FUNCTION_BLOCK FB_McAxisCtrl EXTENDS FB_McAxis IMPLEMENTS I_McAxis
VAR
  _eCheck                   : E_CHECK_STATE;  // pointer check

  _eAxisCycle,                                // cyclic AXIS_REF() and MC_Power check
  _eInit                    : E_PROGRESS;     // axis startup and init, get encoder type, get axis name, get device name

  _nAxisIndex               : UINT;           // know thyself
  _rTargetWindow            : LREAL := 0.1;   // TODO: get that from NC

  // pointers to all; access required for coupling; access by index
  _Axes                     : REFERENCE TO ARRAY[1..PLC_CONSTANT.MAX_AXIS] OF AXIS_REF;

  _Ctrl                     : POINTER TO ARRAY[1..PLC_CONSTANT.MAX_AXIS] OF ST_AXIS_CTRL;    // contains command to be executed
  _State                    : POINTER TO ARRAY[1..PLC_CONSTANT.MAX_AXIS] OF ST_AXIS_STATE;   // mirrors command with added result

  _Info                     : POINTER TO ARRAY[1..PLC_CONSTANT.MAX_AXIS] OF ST_AXIS_INFO;    // axis state and position data to read from
  _Data                     : POINTER TO ARRAY[1..PLC_CONSTANT.MAX_AXIS] OF ST_MOVE_DATA;    // structure for cyclic interface

  _NcParameterWrt           : POINTER TO ARRAY[1..PLC_CONSTANT.MAX_AXIS] OF ST_NC_PARAMETER; // W struct for a single parameter
  _NcParameterRd            : POINTER TO ARRAY[1..PLC_CONSTANT.MAX_AXIS] OF ST_NC_PARAMETER; // R struct for a single parameter
  _HomeParameter            : POINTER TO ARRAY[1..PLC_CONSTANT.MAX_AXIS] OF ST_HOMING;       // homing parameter for each axis

  _GearInParameter          : POINTER TO ARRAY[1..PLC_CONSTANT.MAX_AXIS] OF ST_GEAR_IN;      // Master Indices, dyn constraints for simple GearIn

  _MotionOptions            : POINTER TO ARRAY[1..PLC_CONSTANT.MAX_AXIS] OF ST_MOTION_OPTIONS;


  // local copies of command
  _eCtrl,
  _eCtrlOld                       : E_AXIS_CTRL;

  // Last handled NC Axis parameter to write
  _eParameterNrWrite              : Tc2_MC2.MC_AxisParameter;
  _rParameterWrtValue             : LREAL;

  // Last handled NC Axis parameter to read
  _eParameterNrRead               : Tc2_MC2.MC_AxisParameter;
  _rParameterReadValue            : LREAL;

  // execution state
  _eResult                        : E_PROGRESS;   // result of execution state
  _eResultOld                     : E_PROGRESS;   // old result for detecting change
  _eState                         : E_AXIS_STATE; // execution state

  // calibration options with limit switches and simulation
  _bCalibrationCam                : BOOL;

  // mapping inputs
  _bLimitMin,
  _bLimitMax,
  _bCalibrationInput     AT %I*   : BOOL;


  // placeholder dummies in case count of Multimaster ases <> 4
  {attribute 'hide'}
  _MultiMasterDummyRef            : ARRAY[1..4] OF AXIS_REF;

  _fbGearOut                      : Tc2_MC2.MC_GearOut;
  _fbGearIn                       : Tc2_MC2.MC_GearIn;
  _fbGearInMultiMaster            : Tc2_MC2.MC_GearInMultiMaster;
END_VAR

IF NOT Check() THEN RETURN; END_IF
//-----------------------------------------------------------------------------
// check _HomeParameter for calibration input options
//-----------------------------------------------------------------------------
_bCalibrationCam                    := GetCalibrationCam();
CalibrationCam                      := ADR(_bCalibrationCam);
//-----------------------------------------------------------------------------
//-----------------------------------------------------------------------------
Override                            := _Data^[_nAxisIndex].rOverride;
//-----------------------------------------------------------------------------
//-----------------------------------------------------------------------------
// cyclic call to MC_Power and AXIS_REF()
//-----------------------------------------------------------------------------
_eAxisCycle                         := Cycle();
//-----------------------------------------------------------------------------
//-----------------------------------------------------------------------------
// get command from outside world
//-----------------------------------------------------------------------------
_eCtrl                              := _Ctrl^[_nAxisIndex].eCtrl;
//-----------------------------------------------------------------------------
//-----------------------------------------------------------------------------
//  OnChange react to command
//-----------------------------------------------------------------------------
IF (_eCtrl <> _eCtrlOld)
THEN
  // get busy
  _eState                           := Cmd(_eCtrl); // get execution state for command
  _eCtrlOld                         := _eCtrl;
  LogControl();
END_IF
//-----------------------------------------------------------------------------
//-----------------------------------------------------------------------------
//  execution state for command
//-----------------------------------------------------------------------------
CASE _eState
OF
  E_AXIS_STATE.AXIS_INIT:
    //-------------------------------------------------------------------------
    // axis always requires one init from outside world at startup
    // _eInit has to be valid for other commands to be accepted in Cmd(_eCtrl)
    _eInit := _eResult              := AxisInit(TRUE);

  E_AXIS_STATE.AXIS_NO_INIT:
    //-------------------------------------------------------------------------
    // we are here because you sent a command before having done AXIS_INIT
    _eResult                        := E_PROGRESS.ERROR;

  E_AXIS_STATE.AXIS_DISABLE:
    _eResult                        := AxisDisable(TRUE);

  E_AXIS_STATE.AXIS_ENABLE:
    _eResult                        := AxisEnable(TRUE);

  E_AXIS_STATE.AXIS_IDLE:
    _eResult                        := AxisIdle(TRUE);

  E_AXIS_STATE.AXIS_HOME:
    _eResult                        := AxisHome(TRUE);

  E_AXIS_STATE.AXIS_MOVE_POS:
    _eResult                        := AxisMoveToPosition(TRUE, _Data^[_nAxisIndex]);

  E_AXIS_STATE.AXIS_MOVE_VELO:
    _eResult                        := AxisMoveVelocity(TRUE, _Data^[_nAxisIndex]);

  E_AXIS_STATE.AXIS_RESET:
    _eResult                        := AxisReset(TRUE);

  E_AXIS_STATE.AXIS_HALT:
    _eResult                        := AxisHalt(TRUE, _Data^[_nAxisIndex]);

  E_AXIS_STATE.AXIS_STOP:
    _eResult                        := AxisStop(TRUE, _Data^[_nAxisIndex]);

  E_AXIS_STATE.AXIS_MOVE_BUFFER:
    _eResult                        := AxisBufferPos(TRUE, _Data^[_nAxisIndex]);

  E_AXIS_STATE.AXIS_MOVE_BUFFER_VELO:
    _eResult                        := AxisBufferVelo(TRUE, _Data^[_nAxisIndex]);

  E_AXIS_STATE.AXIS_PARAMETER_READ:
    _eResult                        := AxisParameterRead(TRUE, _NcParameterRd^[_nAxisIndex].ParameterNumber);

  E_AXIS_STATE.AXIS_PARAMETER_WRITE:
    _eResult                        := AxisParameterWrite(TRUE, _NcParameterWrt^[_nAxisIndex].ParameterNumber);

  E_AXIS_STATE.AXIS_PARAMETER_WRITE_PERSISTENT:
    _eResult                        := AxisParameterWritePersistent(TRUE, _NcParameterWrt^[_nAxisIndex].ParameterNumber);

  E_AXIS_STATE.AXIS_GEAR_IN:
    _eResult                        := AxisGearIn(TRUE);

  E_AXIS_STATE.AXIS_GEAR_OUT:
    _eResult                        := AxisGearOut(TRUE);

  E_AXIS_STATE.AXIS_GEAR_IN_MULTIMASTER:
    _eResult                        := AxisGearInMultiMaster(TRUE);

ELSE
  IF (_eCtrl > E_AXIS_CTRL.AXIS_NULL)
  THEN
    _eResult                          := E_PROGRESS.NOT_EXIST;
    _Info^[_nAxisIndex].bError        := TRUE;
  ELSE
    _eResult                          := E_PROGRESS.INVALID;
  END_IF
END_CASE
//-----------------------------------------------------------------------------
//-----------------------------------------------------------------------------
//  OnChange of execution state result
//    - log result and clear error number on interface
//-----------------------------------------------------------------------------
IF (_eResult <> _eResultOld)
THEN
  LogResult();
  _Info^[_nAxisIndex].nErrorId      := 0;
  _eResultOld                       := _eResult;
END_IF
//-----------------------------------------------------------------------------
//-----------------------------------------------------------------------------
// Check AxisInit
//-----------------------------------------------------------------------------
IF NOT (_eInit = E_PROGRESS.DONE)
THEN
  _Info^[_nAxisIndex].bReady        := FALSE;
ELSE
  _Info^[_nAxisIndex].bReady        := _AxisRef.Status.ControlLoopClosed AND
                                       (NOT _AxisRef.Status.Error)       AND 
                                       (NOT _AxisRef.Status.Moving);
END_IF
//-----------------------------------------------------------------------------
//  execution state result error
//-----------------------------------------------------------------------------
CASE _eResult
OF
  E_PROGRESS.ERROR:
    _Info^[_nAxisIndex].bReady      := FALSE;
    _Info^[_nAxisIndex].bError      := TRUE;
    _Info^[_nAxisIndex].nErrorId    := ErrorId;
END_CASE
//-----------------------------------------------------------------------------
// execution state result to interface
//-----------------------------------------------------------------------------
_State^[_nAxisIndex].eState       := _eState + _eResult;
//-----------------------------------------------------------------------------
// encoder type (enum)
//-----------------------------------------------------------------------------
_State^[_nAxisIndex].eAxisEncoder := EncoderType;
//-----------------------------------------------------------------------------
// _stState.[nAxisIndex].eState is overridden by MC_Power.bError
//  _eAxisCycle := Cycle() is called at the top; checks MC_Power.bError
//  MC_Power.bError requires e_AXIS_CTRL.AXIS_RESET in order to clear
//-----------------------------------------------------------------------------
CASE _eAxisCycle
OF
  E_PROGRESS.ERROR:
    _Info^[_nAxisIndex].bReady      := FALSE;
    _Info^[_nAxisIndex].bError      := TRUE;
    _State^[_nAxisIndex].eState   := _eState + _eAxisCycle;
END_CASE
//-----------------------------------------------------------------------------
// Check ControlLoop
//-----------------------------------------------------------------------------
IF _AxisRef.Status.ControlLoopClosed
THEN
  _Info^[_nAxisIndex].bEnabled      := TRUE;
ELSE
  _Info^[_nAxisIndex].bEnabled      := FALSE;
END_IF
//-----------------------------------------------------------------------------
_Info^[_nAxisIndex].bStandstill     := _AxisRef.Status.NotMoving;
//-----------------------------------------------------------------------------
_Info^[_nAxisIndex].rActPos         := _AxisRef.NcToPlc.ActPos;
_Info^[_nAxisIndex].rActVelo        := _AxisRef.NcToPlc.ActVelo;
_Info^[_nAxisIndex].rPosDiff        := _AxisRef.NcToPlc.PosDiff;
//-----------------------------------------------------------------------------
IF (_Info^[_nAxisIndex].rActPos < _Data^[_nAxisIndex].rSetPos + _rTargetWindow) AND
   (_Info^[_nAxisIndex].rActPos > _Data^[_nAxisIndex].rSetPos - _rTargetWindow) AND
    _Info^[_nAxisIndex].bStandstill
THEN
  _Info^[_nAxisIndex].bInTarget     := TRUE;
ELSE
  _Info^[_nAxisIndex].bInTarget     := FALSE;
END_IF
//-----------------------------------------------------------------------------
// copy CoupleState from axis
//-----------------------------------------------------------------------------
_Info^[_nAxisIndex].dwCoupleState   := _AxisRef.NcToPlc.CoupleState;
//-----------------------------------------------------------------------------
//-----------------------------------------------------------------------------
// copy NC AxisId from axis
//-----------------------------------------------------------------------------
_Info^[_nAxisIndex].nNcAxisId       := _AxisRef.NcToPlc.AxisId;
//-----------------------------------------------------------------------------

PROPERTY Axes : reference TO ARRAY[1..PLC_CONSTANT.MAX_AXIS] OF AXIS_REF
SET
_Axes := Axes;
END_SET
END_PROPERTY

METHOD AxisBufferPos : E_PROGRESS
VAR_INPUT
  Enable            : BOOL;
  Data              : ST_MOVE_DATA;
END_VAR
VAR_INST
  _BufferMode       : Tc2_MC2.MC_BufferMode;
  _eres,
  _eState           : E_PROGRESS;
END_VAR
IF NOT Check() THEN AxisBufferPos := E_PROGRESS.ERROR; RETURN; END_IF
IF NOT Enable THEN _eState := E_PROGRESS.INIT; END_IF

CASE _eState
OF
  E_PROGRESS.INIT:
    IF Enable 
    THEN
      _eState       := E_PROGRESS.BUSY;
    END_IF
END_CASE
CASE _eState
OF
  E_PROGRESS.BUSY:
    _eState         := E_PROGRESS.WORKING;
    _BufferMode     := _MotionOptions^[_nAxisIndex].eBufferMode;
    _eres           := MovePosBuffer(
                                  Enable      := FALSE, 
                                  Position    := Data.rSetPos, 
                                  Vel         := Data.rSetVelo, 
                                  Acc         := Data.rAcc, 
                                  Dec         := Data.rDec, 
                                  Jerk        := Data.rJerk, 
                                  BufferMode  := _BufferMode);
END_CASE
CASE _eState
OF
  E_PROGRESS.WORKING:
    _BufferMode     := _MotionOptions^[_nAxisIndex].eBufferMode;
    _eres           := MovePosBuffer(
                                  Enable      := TRUE, 
                                  Position    := Data.rSetPos, 
                                  Vel         := Data.rSetVelo, 
                                  Acc         := Data.rAcc, 
                                  Dec         := Data.rDec, 
                                  Jerk        := Data.rJerk, 
                                  BufferMode  := _BufferMode);
    IF (_eres = E_PROGRESS.ERROR)
    THEN
      _eState       := E_PROGRESS.ERROR;
                       MovePosBuffer(
                                  Enable      := FALSE, 
                                  Position    := Data.rSetPos, 
                                  Vel         := Data.rSetVelo, 
                                  Acc         := Data.rAcc, 
                                  Dec         := Data.rDec, 
                                  Jerk        := Data.rJerk, 
                                  BufferMode  := _BufferMode);

    ELSIF (_Ctrl^[_nAxisIndex].eProgress = E_PROGRESS.DONE)
    THEN
      // when Ctrl decides to leave; make finishing move and be done
      _eState       := E_PROGRESS.FINISHING;
    END_IF
END_CASE
CASE _eState
OF
  E_PROGRESS.FINISHING:
    _eState         := E_PROGRESS.DONE;
    _eres           := MovePosBuffer(
                                  Enable      := FALSE, 
                                  Position    := Data.rSetPos, 
                                  Vel         := Data.rSetVelo, 
                                  Acc         := Data.rAcc, 
                                  Dec         := Data.rDec, 
                                  Jerk        := Data.rJerk, 
                                  BufferMode  := _BufferMode);
END_CASE

AxisBufferPos       := _eState;
END_METHOD

METHOD AxisBufferVelo : E_PROGRESS
VAR_INPUT
  Enable            : BOOL;
  Data              : ST_MOVE_DATA;
END_VAR
VAR_INST
  _BufferMode       : Tc2_MC2.MC_BufferMode;
  _eres,
  _eState           : E_PROGRESS;
END_VAR
IF NOT Check() THEN AxisBufferVelo := E_PROGRESS.ERROR; RETURN; END_IF
IF NOT Enable THEN _eState := E_PROGRESS.INIT; END_IF

CASE _eState
OF
  E_PROGRESS.INIT:
    IF Enable 
    THEN
      _eState       := E_PROGRESS.BUSY;
    END_IF
END_CASE
CASE _eState
OF
  E_PROGRESS.BUSY:
    _eState         := E_PROGRESS.WORKING;
    _BufferMode     := _MotionOptions^[_nAxisIndex].eBufferMode;
    _eres           := MoveVeloBuffer(
                                  Enable      := FALSE, 
                                  Velocity    := Data.rSetVelo, 
                                  Acc         := Data.rAcc, 
                                  Dec         := Data.rDec, 
                                  Jerk        := Data.rJerk, 
                                  BufferMode  := _BufferMode);

END_CASE
CASE _eState
OF
  E_PROGRESS.WORKING:
    _BufferMode     := _MotionOptions^[_nAxisIndex].eBufferMode;
    _eres           := MoveVeloBuffer(
                                  Enable      := TRUE, 
                                  Velocity    := Data.rSetVelo, 
                                  Acc         := Data.rAcc, 
                                  Dec         := Data.rDec, 
                                  Jerk        := Data.rJerk, 
                                  BufferMode  := _BufferMode);
    IF (_eres = E_PROGRESS.ERROR)
    THEN
      _eState := E_PROGRESS.ERROR;
                       MoveVeloBuffer(
                                  Enable      := FALSE, 
                                  Velocity    := Data.rSetVelo, 
                                  Acc         := Data.rAcc, 
                                  Dec         := Data.rDec, 
                                  Jerk        := Data.rJerk, 
                                  BufferMode  := _BufferMode);

    ELSIF (_Ctrl^[_nAxisIndex].eProgress = E_PROGRESS.DONE)
    THEN
      // when Ctrl decides to leave; make finishing move and be done
      _eState       := E_PROGRESS.FINISHING;
    END_IF
END_CASE
CASE _eState
OF
  E_PROGRESS.FINISHING:
    _eState         := E_PROGRESS.DONE;
    _eres           := MoveVeloBuffer(
                                  Enable      := FALSE, 
                                  Velocity    := Data.rSetVelo, 
                                  Acc         := Data.rAcc, 
                                  Dec         := Data.rDec, 
                                  Jerk        := Data.rJerk, 
                                  BufferMode  := _BufferMode);
END_CASE

AxisBufferVelo      := _eState;
END_METHOD

PROPERTY AxisCtrl : pointer to ARRAY[1..PLC_CONSTANT.MAX_AXIS] OF st_axis_ctrl
SET
_Ctrl := AxisCtrl;
END_SET
END_PROPERTY

PROPERTY AxisData : pointer to ARRAY[1..PLC_CONSTANT.MAX_AXIS] OF st_move_data
SET
_Data := AxisData;
END_SET
END_PROPERTY

METHOD AxisDisable : E_PROGRESS
VAR_INPUT
  Execute           : BOOL;
END_VAR
VAR_INST
  _eState,
  _eResult          : E_PROGRESS;
  _rValue           : LREAL;
  _udiErr           : UDINT;
  _stMsg            : ST_Message;


END_VAR
IF NOT Check() THEN AxisDisable := E_PROGRESS.ERROR; RETURN; END_IF
IF NOT Execute THEN _eState := E_PROGRESS.INIT; END_IF

CASE _eState
OF
  E_PROGRESS.INIT:
    IF Execute 
    THEN
      memset(ADR(_stMsg),0,SIZEOF(_stMsg));
      _udiErr                       := 0;
      _rValue                       := 0;
      _eState                       := E_PROGRESS.BUSY;
    END_IF
END_CASE
CASE _eState
OF
  E_PROGRESS.BUSY:
    _eResult                        := Disable(FALSE);
    _eState                         := E_PROGRESS.WAITING;
END_CASE
CASE _eState
OF
  E_PROGRESS.WAITING:
    _eResult                        := Disable(TRUE);

    IF (_eResult = E_PROGRESS.DONE)
    THEN
      _eState                       := E_PROGRESS.WORKING;
    END_IF
END_CASE
CASE _eState
OF
  E_PROGRESS.WORKING:
    _eState                         := E_PROGRESS.DONE;
END_CASE

AxisDisable := _eState;
END_METHOD

METHOD AxisEnable : E_PROGRESS
VAR_INPUT
  Execute           : BOOL;
END_VAR
VAR_INST
  _eState,
  _eResult          : E_PROGRESS;
  _rValue           : LREAL;
  _udiErr           : UDINT;
  _stMsg            : ST_Message;


END_VAR
IF NOT Check() THEN AxisEnable := E_PROGRESS.ERROR; RETURN; END_IF
IF NOT Execute THEN _eState := E_PROGRESS.INIT; END_IF

CASE _eState
OF
  E_PROGRESS.INIT:
    IF Execute 
    THEN
      memset(ADR(_stMsg),0,SIZEOF(_stMsg));
      _udiErr                       := 0;
      _rValue                       := 0;
      _eState                       := E_PROGRESS.BUSY;
    END_IF
END_CASE
CASE _eState
OF
  E_PROGRESS.BUSY:
    _eResult                        := Enable(FALSE);
    _eState                         := E_PROGRESS.WAITING;
END_CASE
CASE _eState
OF
  E_PROGRESS.WAITING:
    _eResult                        := Enable(TRUE);

    IF (_eResult = E_PROGRESS.DONE)
    THEN
      _eState                       := E_PROGRESS.WORKING;
    END_IF
END_CASE
CASE _eState
OF
  E_PROGRESS.WORKING:
    _eState                         := E_PROGRESS.DONE;
END_CASE

AxisEnable := _eState;
END_METHOD

METHOD AxisGearIn : E_PROGRESS
VAR_INPUT
  Execute           : BOOL;
END_VAR
VAR_INST
  _eState           : E_PROGRESS;
  _rValue           : LREAL;
  _nErr,
  _nMasterIndex,
  _nMasterNcId      : UDINT;
  _stMsg            : ST_Message;


END_VAR
IF NOT Check() THEN AxisGearIn := E_PROGRESS.ERROR; RETURN; END_IF
IF NOT Execute THEN _eState := E_PROGRESS.INIT; END_IF

CASE _eState
OF
  E_PROGRESS.INIT:
    IF Execute 
    THEN
      memset(ADR(_stMsg),0,SIZEOF(_stMsg));
      _nMasterNcId                  :=
      _nMasterIndex                 :=
      _nErr                         := 0;
      _rValue                       := 0;

      IF NOT (_GearInParameter^[_nAxisIndex].nAxisIndexMaster[1] > 0) OR
         NOT (_GearInParameter^[_nAxisIndex].nAxisIndexMaster[1] < MAX_AXIS+1)
      THEN
        _nMasterIndex               := _GearInParameter^[_nAxisIndex].nAxisIndexMaster[1];

        _stMsg.eType                := E_MessageType.eMessageError;
        _stMsg.eDevice              := e_Device.Axis + TO_UINT(_AxisRef.NcToPlc.AxisId);
        _stMsg.eSubdevice           := e_Subdevice.fbGearIn;
        _stMsg.iErrorNumber         := 
        _nErr                       := 666;

        _stMsg.sText                := concat('_GearInParameter[', TO_STRING(_nAxisIndex));
        _stMsg.sText                := concat(_stMsg.sText,    '].nAxisIndexMaster[1] out of range: ');
        _stMsg.sText                := concat(_stMsg.sText, TO_STRING(_nMasterIndex));

        f_MessageSet(_stMsg);

        _eState                     := E_PROGRESS.ERROR;

      ELSE
        _eState                     := E_PROGRESS.BUSY;

        _nMasterIndex               := _GearInParameter^[_nAxisIndex].nAxisIndexMaster[1];
        _nMasterNcId                := _Info^[_nMasterIndex].nNcAxisId;

        _stMsg.eType                := E_MessageType.eMessageInfo;
        _stMsg.eDevice              := e_Device.Axis + TO_UINT(_AxisRef.NcToPlc.AxisId);
        _stMsg.eSubdevice           := e_Subdevice.fbGearIn;
        _stMsg.iErrorNumber         := 0;
  
        _stMsg.sText                := concat('GearIn BUSY: ', TO_STRING(_nMasterIndex));
        f_MessageSet(_stMsg);
      END_IF
    END_IF
END_CASE
CASE _eState
OF
  E_PROGRESS.BUSY:
    _eState                         := E_PROGRESS.STARTUP;
    _fbGearIn(
              Master                := _Axes[_nMasterIndex], 
              Slave                 := _AxisRef, 
              Execute               := FALSE, 
              RatioNumerator        := _GearInParameter^[_nAxisIndex].rGearRatio[1], 
              RatioDenominator      := 1, 
              Acceleration          := _GearInParameter^[_nAxisIndex].Acceleration, 
              Deceleration          := _GearInParameter^[_nAxisIndex].Deceleration, 
              Jerk                  := _GearInParameter^[_nAxisIndex].Jerk);
END_CASE
CASE _eState
OF
  E_PROGRESS.STARTUP:
    _fbGearIn(
              Master                := _Axes[_nMasterIndex], 
              Slave                 := _AxisRef, 
              Execute               := TRUE, 
              RatioNumerator        := _GearInParameter^[_nAxisIndex].rGearRatio[1], 
              RatioDenominator      := 1, 
              Acceleration          := _GearInParameter^[_nAxisIndex].Acceleration, 
              Deceleration          := _GearInParameter^[_nAxisIndex].Deceleration, 
              Jerk                  := _GearInParameter^[_nAxisIndex].Jerk);

    IF (_fbGearIn.Error)
    THEN
      _nErr                         := _fbGearIn.ErrorID;

      _stMsg.eType                  := E_MessageType.eMessageError;
      _stMsg.eDevice                := e_Device.Axis + TO_UINT(_AxisRef.NcToPlc.AxisId);
      _stMsg.eSubdevice             := e_Subdevice.fbGearIn;
      _stMsg.iErrorNumber           := _nErr;

      _stMsg.sText                  := concat('GearIn ERROR: ', TO_STRING(_nMasterIndex));
      f_MessageSet(_stMsg);
      _eState                       := E_PROGRESS.ERROR;

    ELSIF (_fbGearIn.InGear)
    THEN
      _eState                       := E_PROGRESS.READY;
    END_IF
END_CASE
CASE _eState
OF
  E_PROGRESS.READY:
    _eState                         := E_PROGRESS.DONE;

    _stMsg.eType                    := E_MessageType.eMessageInfo;
    _stMsg.eDevice                  := e_Device.Axis + TO_UINT(_AxisRef.NcToPlc.AxisId);
    _stMsg.eSubdevice               := e_Subdevice.fbGearIn;
    _stMsg.iErrorNumber             := 0;

    _stMsg.sText                    := concat('GearIn done: ', TO_STRING(_nMasterIndex));
    f_MessageSet(_stMsg);
END_CASE
CASE _eState
OF
  E_PROGRESS.DONE,
  E_PROGRESS.ERROR:
    _fbGearIn(
              Master                := _Axes[_nMasterIndex], 
              Slave                 := _AxisRef, 
              Execute               := FALSE);
END_CASE

AxisGearIn                          := _eState;
END_METHOD

METHOD AxisGearInMultiMaster : E_PROGRESS
VAR_INPUT
  Execute           : BOOL;
END_VAR
VAR_INST
  _eState           : E_PROGRESS;
  _rValue           : LREAL;
  _nAx,
  _nErr             : UDINT;

  _nMasterIndex,
  _nMasterNcId      : ARRAY[1..4] OF UDINT;

  _stOptions        : Tc2_MC2.ST_GearInMultiMasterOptions;
  _nSyncMode        : int;

  _stMsg            : ST_Message;


END_VAR
IF NOT Check() THEN AxisGearInMultiMaster := E_PROGRESS.ERROR; RETURN; END_IF
IF NOT Execute THEN _eState := E_PROGRESS.INIT; END_IF

CASE _eState
OF
  E_PROGRESS.INIT:
    IF Execute 
    THEN
      memset(ADR(_stMsg),0,SIZEOF(_stMsg));
      memset(ADR(_nMasterNcId), 0,SIZEOF(_nMasterNcId));
      memset(ADR(_nMasterIndex),0,SIZEOF(_nMasterIndex));
      memset(ADR(_stOptions),   0,SIZEOF(_stOptions));
      _nErr                           := 0;
      _rValue                         := 0;

      IF NOT (_GearInParameter^[_nAxisIndex].nAxisIndexMaster[1] > 0) OR
         NOT (_GearInParameter^[_nAxisIndex].nAxisIndexMaster[1] <= MAX_AXIS)
      THEN
        _nMasterIndex[1]              := _GearInParameter^[_nAxisIndex].nAxisIndexMaster[1];

        _stMsg.eType                  := E_MessageType.eMessageError;
        _stMsg.eDevice                := e_Device.Axis + TO_UINT(_AxisRef.NcToPlc.AxisId);
        _stMsg.eSubdevice             := e_Subdevice.fbGearInMultiMaster;
        _stMsg.iErrorNumber           := 
        _nErr                         := 666;

        _stMsg.sText                  := concat('_GearInParameter[', TO_STRING(_nAxisIndex));
        _stMsg.sText                  := concat(_stMsg.sText,    '].nAxisIndexMaster[1] out of range: ');
        _stMsg.sText                  := concat(_stMsg.sText, TO_STRING(_nMasterIndex[1]));
        f_MessageSet(_stMsg);

        _eState                       := E_PROGRESS.ERROR;

      ELSE
        _eState                       := E_PROGRESS.BUSY;

        _stOptions.AdvancedSlaveDynamics  := _GearInParameter^[_nAxisIndex].bAdvancedSlaveDynamics;
        _nSyncMode                        := _GearInParameter^[_nAxisIndex].nMultiMasterSyncMode;

        _nMasterIndex[1]              := _GearInParameter^[_nAxisIndex].nAxisIndexMaster[1];
        _nMasterNcId[1]               := _Info^[_nMasterIndex[1]].nNcAxisId;
        memcpy(ADR(_stOptions.SyncMode), ADR(_nSyncMode), SIZEOF(_stOptions.SyncMode));

        _fbGearInMultiMaster.Master1  := _Axes[_nMasterIndex[1]];   // assign AXIS_REF of master

        _stMsg.eType                  := E_MessageType.eMessageInfo;
        _stMsg.eDevice                := e_Device.Axis + TO_UINT(_AxisRef.NcToPlc.AxisId);
        _stMsg.eSubdevice             := e_Subdevice.fbGearInMultiMaster;
        _stMsg.iErrorNumber           := _eState;

        _stMsg.sText                  := concat('_GearInParameter[', TO_STRING(_nAxisIndex));
        _stMsg.sText                  := concat(_stMsg.sText,    '] MultiMaster check: ');
        _stMsg.sText                  := concat(_stMsg.sText, TO_STRING(_nMasterIndex[1]));
        f_MessageSet(_stMsg);

        _nAx                          := 2; // next master index to check
      END_IF
    END_IF
END_CASE
CASE _eState
OF
  E_PROGRESS.BUSY:
    IF NOT (_GearInParameter^[_nAxisIndex].nAxisIndexMaster[_nAx] > 0) OR
       NOT (_GearInParameter^[_nAxisIndex].nAxisIndexMaster[_nAx] < MAX_AXIS+1)
    THEN
      // next entry not valid
      // Master1 is already checked --> let's get ready
      _eState                         := E_PROGRESS.READY;
    ELSE
      _eState                         := E_PROGRESS.STARTUP;

      _nMasterIndex[_nAx]             := _GearInParameter^[_nAxisIndex].nAxisIndexMaster[_nAx];
      _nMasterNcId [_nAx]             := _Info^[_nMasterIndex[_nAx]].nNcAxisId;

      _stMsg.eType                    := E_MessageType.eMessageInfo;
      _stMsg.eDevice                  := e_Device.Axis + TO_UINT(_AxisRef.NcToPlc.AxisId);
      _stMsg.eSubdevice               := e_Subdevice.fbGearInMultiMaster;
      _stMsg.iErrorNumber             := _eState;

      _stMsg.sText                    := concat('_GearInParameter[', TO_STRING(_nAxisIndex));
      _stMsg.sText                    := concat(_stMsg.sText,    '] MultiMaster check: ');
      _stMsg.sText                    := concat(_stMsg.sText, TO_STRING(_nMasterIndex[_nAx]));
      f_MessageSet(_stMsg);
    END_IF

    _fbGearInMultiMaster(
                      Slave           := _AxisRef, 
                      Enable          := FALSE, 
                      GearRatio1      := _GearInParameter^[_nAxisIndex].rGearRatio[1], 
                      GearRatio2      := _GearInParameter^[_nAxisIndex].rGearRatio[2], 
                      GearRatio3      := _GearInParameter^[_nAxisIndex].rGearRatio[3], 
                      GearRatio4      := _GearInParameter^[_nAxisIndex].rGearRatio[4], 
                      Acceleration    := _GearInParameter^[_nAxisIndex].Acceleration, 
                      Deceleration    := _GearInParameter^[_nAxisIndex].Deceleration, 
                      Jerk            := _GearInParameter^[_nAxisIndex].Jerk,
                      Options         := _stOptions);
END_CASE
CASE _eState
OF
  E_PROGRESS.STARTUP:
    CASE _nAx
    OF
      2:
        _nAx                          := _nAx + 1;
        _eState                       := E_PROGRESS.BUSY;
        _fbGearInMultiMaster.Master2  := _Axes[_nMasterIndex[2]];   // assign AXIS_REF of master

      3:
        _nAx                          := _nAx + 1;
        _eState                       := E_PROGRESS.BUSY;
        _fbGearInMultiMaster.Master3  := _Axes[_nMasterIndex[3]];   // assign AXIS_REF of master

      4:
        _nAx                          := _nAx + 1;
        _eState                       := E_PROGRESS.BUSY;
        _fbGearInMultiMaster.Master4  := _Axes[_nMasterIndex[4]];   // assign AXIS_REF of master
    ELSE
      _eState                         := E_PROGRESS.READY;
    END_CASE
END_CASE
CASE _eState
OF
  E_PROGRESS.READY:
    _fbGearInMultiMaster(
                      Slave           := _AxisRef, 
                      Enable          := TRUE, 
                      GearRatio1      := _GearInParameter^[_nAxisIndex].rGearRatio[1], 
                      GearRatio2      := _GearInParameter^[_nAxisIndex].rGearRatio[2], 
                      GearRatio3      := _GearInParameter^[_nAxisIndex].rGearRatio[3], 
                      GearRatio4      := _GearInParameter^[_nAxisIndex].rGearRatio[4], 
                      Acceleration    := _GearInParameter^[_nAxisIndex].Acceleration, 
                      Deceleration    := _GearInParameter^[_nAxisIndex].Deceleration, 
                      Jerk            := _GearInParameter^[_nAxisIndex].Jerk);

    IF (_fbGearInMultiMaster.Error)
    THEN
      _nErr                           := _fbGearInMultiMaster.ErrorID;
      _stMsg.eType                    := E_MessageType.eMessageError;
      _stMsg.eDevice                  := e_Device.Axis + TO_UINT(_AxisRef.NcToPlc.AxisId);
      _stMsg.eSubdevice               := e_Subdevice.fbGearInMultiMaster;
      _stMsg.iErrorNumber             := _nErr;

      _stMsg.sText                    := concat(TO_STRING(_eCtrl),'[');
      _stMsg.sText                    := concat(_stMsg.sText, TO_STRING(_nAxisIndex));
      _stMsg.sText                    := concat(_stMsg.sText, ']');
      _stMsg.sText                    := concat('fbGearInMultiMaster error: ', TO_STRING(_nErr));
      f_MessageSet(_stMsg);
      _eState                         := E_PROGRESS.ERROR;

    ELSIF (_fbGearIn.InGear)
    THEN
      _eState                         := E_PROGRESS.WORKING;
    END_IF

END_CASE
CASE _eState
OF
  E_PROGRESS.WORKING:
    // now GearRatio[x] can be altered from outside
    // axis function waits here for further instructions from outside world
    // _stCtrl[_nAxisIndex].eProgress = e_Progress.DONE must be used to leave this axis function
    _fbGearInMultiMaster(
                      Slave           := _AxisRef, 
                      Enable          := TRUE, 
                      GearRatio1      := _GearInParameter^[_nAxisIndex].rGearRatio[1], 
                      GearRatio2      := _GearInParameter^[_nAxisIndex].rGearRatio[2], 
                      GearRatio3      := _GearInParameter^[_nAxisIndex].rGearRatio[3], 
                      GearRatio4      := _GearInParameter^[_nAxisIndex].rGearRatio[4], 
                      Acceleration    := _GearInParameter^[_nAxisIndex].Acceleration, 
                      Deceleration    := _GearInParameter^[_nAxisIndex].Deceleration, 
                      Jerk            := _GearInParameter^[_nAxisIndex].Jerk);

    IF (_fbGearInMultiMaster.Error)
    THEN
      _nErr                           := _fbGearInMultiMaster.ErrorID;
      _stMsg.eType                    := E_MessageType.eMessageError;
      _stMsg.eDevice                  := e_Device.Axis + TO_UINT(_AxisRef.NcToPlc.AxisId);
      _stMsg.eSubdevice               := e_Subdevice.fbGearInMultiMaster;
      _stMsg.iErrorNumber             := _nErr;

      _stMsg.sText                    := concat(TO_STRING(_eCtrl),'[');
      _stMsg.sText                    := concat(_stMsg.sText, TO_STRING(_nAxisIndex));
      _stMsg.sText                    := concat(_stMsg.sText, ']');
      _stMsg.sText                    := concat('fbGearInMultiMaster error: ', TO_STRING(_nErr));
      f_MessageSet(_stMsg);
      _eState                         := E_PROGRESS.ERROR;

    ELSIF (_Ctrl^[_nAxisIndex].eProgress = E_PROGRESS.DONE)
    THEN
      // when Ctrl decides to leave; make finishing move and be done
      _eState                         := E_PROGRESS.FINISHING;
    END_IF
END_CASE
CASE _eState
OF
  E_PROGRESS.FINISHING:
    _eState                           := E_PROGRESS.DONE;

    _stMsg.eType                      := E_MessageType.eMessageInfo;
    _stMsg.eDevice                    := e_Device.Axis + TO_UINT(_AxisRef.NcToPlc.AxisId);
    _stMsg.eSubdevice                 := e_Subdevice.fbGearInMultiMaster;
    _stMsg.iErrorNumber               := _eState;

    _stMsg.sText                      := concat(TO_STRING(_eCtrl), ': ');
    _stMsg.sText                      := concat(_stMsg.sText, TO_STRING(_eState));
    f_MessageSet(_stMsg);
END_CASE

AxisGearInMultiMaster                 := _eState;
END_METHOD

PROPERTY AxisGearInParameter : pointer to ARRAY[1..PLC_CONSTANT.MAX_AXIS] OF ST_GEAR_IN
SET
_GearInParameter := AxisGearInParameter;
END_SET
END_PROPERTY

METHOD AxisGearOut : E_PROGRESS
VAR_INPUT
  Execute           : BOOL;
END_VAR
VAR_INST
  _eState           : E_PROGRESS;
  _rValue           : LREAL;
  _nErr             : UDINT;
  _stMsg            : ST_Message;
END_VAR
IF NOT Check() THEN AxisGearOut := E_PROGRESS.ERROR; RETURN; END_IF
IF NOT Execute THEN _eState := E_PROGRESS.INIT; END_IF

CASE _eState
OF
  E_PROGRESS.INIT:
    IF Execute 
    THEN
      memset(ADR(_stMsg),0,SIZEOF(_stMsg));
      _nErr                       := 0;
      _rValue                     := 0;

      _fbGearOut(
            Slave                 := _AxisRef, 
            Execute               := FALSE);

      IF (_AxisRef.NcToPlc.CoupleState < 2)
      THEN
        _eState                   := E_PROGRESS.DONE;
      ELSE
        _eState                   := E_PROGRESS.BUSY;

        _stMsg.eType              := E_MessageType.eMessageInfo;
        _stMsg.eDevice            := e_Device.Axis + TO_UINT(_AxisRef.NcToPlc.AxisId);
        _stMsg.eSubdevice         := e_Subdevice.fbGearOut;
        _stMsg.iErrorNumber       := 0;
  
        _stMsg.sText              := concat('GearOut BUSY: ', TO_STRING(_nAxisIndex));
        f_MessageSet(_stMsg);
      END_IF
    END_IF
END_CASE
CASE _eState
OF
  E_PROGRESS.BUSY:
    _fbGearOut(
            Slave                 := _AxisRef, 
            Execute               := TRUE);

    IF (_fbGearOut.Error)
    THEN
      _nErr                       := _fbGearOut.ErrorID;

      _stMsg.eType                := E_MessageType.eMessageError;
      _stMsg.eDevice              := e_Device.Axis + TO_UINT(_AxisRef.NcToPlc.AxisId);
      _stMsg.eSubdevice           := e_Subdevice.fbGearOut;
      _stMsg.iErrorNumber         := _nErr;

      _stMsg.sText                := concat('GearOut ERROR: ', TO_STRING(_nAxisIndex));
      f_MessageSet(_stMsg);
      _eState                     := E_PROGRESS.ERROR;

    ELSIF (_fbGearOut.Done)
    THEN
      _stMsg.eType                := E_MessageType.eMessageInfo;
      _stMsg.eDevice              := e_Device.Axis + TO_UINT(_AxisRef.NcToPlc.AxisId);
      _stMsg.eSubdevice           := e_Subdevice.fbGearOut;
      _stMsg.iErrorNumber         := 0;
  
      _stMsg.sText                := concat('GearOut DONE: ', TO_STRING(_nAxisIndex));
      f_MessageSet(_stMsg);

      IF (_AxisRef.NcToPlc.CoupleState < 2)
      THEN
        _eState                   := E_PROGRESS.DONE;
      ELSE
        _eState                   := E_PROGRESS.STARTUP;
      END_IF
    END_IF
END_CASE
CASE _eState
OF
  E_PROGRESS.STARTUP:
    _eState                       := E_PROGRESS.BUSY;
    _fbGearOut(
          Slave                   := _AxisRef, 
          Execute                 := FALSE);

    _stMsg.eType                  := E_MessageType.eMessageInfo;
    _stMsg.eDevice                := e_Device.Axis + TO_UINT(_AxisRef.NcToPlc.AxisId);
    _stMsg.eSubdevice             := e_Subdevice.fbGearOut;
    _stMsg.iErrorNumber           := 0;

    _stMsg.sText                  := concat('GearOut CoupleState: ', TO_STRING(_AxisRef.NcToPlc.CoupleState));
    f_MessageSet(_stMsg);
END_CASE
CASE _eState
OF
  E_PROGRESS.DONE,
  E_PROGRESS.ERROR:
    _fbGearOut(
            Slave                 := _AxisRef, 
            Execute               := FALSE);
END_CASE

AxisGearOut                       := _eState;
END_METHOD

METHOD AxisHalt : E_PROGRESS
VAR_INPUT
  Execute           : BOOL;
  Data              : ST_MOVE_DATA;
END_VAR
VAR_INST
  _eres,
  _eState           : E_PROGRESS;
  _rValue           : LREAL;
  _udiErr           : UDINT;
  _stMsg            : ST_Message;


END_VAR
IF NOT Check() THEN AxisHalt := E_PROGRESS.ERROR; RETURN; END_IF
IF NOT Execute THEN _eState := E_PROGRESS.INIT; END_IF

CASE _eState
OF
  E_PROGRESS.INIT:
    IF Execute 
    THEN
      memset(ADR(_stMsg),0,SIZEOF(_stMsg));
      _udiErr       := 0;
      _rValue       := 0;
      _eState       := E_PROGRESS.BUSY;
    END_IF
END_CASE
CASE _eState
OF
  E_PROGRESS.BUSY:
    _eState         := E_PROGRESS.WAITING;
    _eres           := Halt(
                            Execute := FALSE, 
                            Dec     := Data.rDec, 
                            Jerk    := Data.rJerk);
END_CASE
CASE _eState
OF
  E_PROGRESS.WAITING:
    _eres           := Halt(
                            Execute := TRUE, 
                            Dec     := Data.rDec, 
                            Jerk    := Data.rJerk);

    IF (_eres = E_PROGRESS.ERROR)
    THEN
        _eState     := E_PROGRESS.ERROR;
    ELSIF (_eres = E_PROGRESS.DONE)
    THEN 
      _eState       := E_PROGRESS.WORKING;
    END_IF
END_CASE
CASE _eState
OF
  E_PROGRESS.WORKING:
    _eState         := E_PROGRESS.DONE;
    _eres           := Halt(
                            Execute := FALSE, 
                            Dec     := Data.rDec, 
                            Jerk    := Data.rJerk);
END_CASE

AxisHalt := _eState;
END_METHOD

METHOD AxisHome : E_PROGRESS
VAR_INPUT
  Execute           : BOOL;
END_VAR
VAR_INST
  _eres,
  _eState           : E_PROGRESS;
  _rValue           : LREAL;
  _udiErr           : UDINT;
  _stMsg            : ST_Message;


END_VAR
IF NOT Check() THEN AxisHome := E_PROGRESS.ERROR; RETURN; END_IF
IF NOT Execute THEN _eState := E_PROGRESS.INIT; END_IF

CASE _eState
OF
  E_PROGRESS.INIT:
    IF Execute 
    THEN
      memset(ADR(_stMsg),0,SIZEOF(_stMsg));
      _udiErr               := 0;
      _rValue               := 0;

      IF (_AxisRef.Status.Homed)
      THEN
        _eState             := E_PROGRESS.BUSY;
      ELSE
        _eState             := E_PROGRESS.PREPARE;
      END_IF
    END_IF
END_CASE
CASE _eState
OF
  E_PROGRESS.BUSY:
    _eState                 := E_PROGRESS.STARTUP;
    _eres                   := Home(Execute   := FALSE,
                                    Position  := _HomeParameter^[_nAxisIndex].stHomingParam.Position,
                                    HomingMode:= Tc2_MC2.MC_HomingMode.MC_ResetCalibration,
                                    Options   := _HomeParameter^[_nAxisIndex].stHomingParam.Options);

END_CASE
CASE _eState
OF
  E_PROGRESS.STARTUP:
    _Info^[_nAxisIndex].bReferenced   := FALSE;

    _eres                   := Home(
                                    Execute   := TRUE,
                                    Position  := _HomeParameter^[_nAxisIndex].stHomingParam.Position,
                                    HomingMode:= Tc2_MC2.MC_HomingMode.MC_ResetCalibration,
                                    Options   := _HomeParameter^[_nAxisIndex].stHomingParam.Options);
    IF (_eres = E_PROGRESS.DONE)
    THEN
      _eState               := E_PROGRESS.PREPARE;
    END_IF
END_CASE
CASE _eState
OF
  E_PROGRESS.PREPARE:
      _eState               := E_PROGRESS.READY;

      _eres                 := Home(
                                    Execute   := FALSE,
                                    Position  := _HomeParameter^[_nAxisIndex].stHomingParam.Position,
                                    HomingMode:= Tc2_MC2.MC_HomingMode.MC_ResetCalibration,
                                    Options   := _HomeParameter^[_nAxisIndex].stHomingParam.Options);
END_CASE
CASE _eState
OF
  E_PROGRESS.READY:
    _eState                 := E_PROGRESS.WAITING;

END_CASE
CASE _eState
OF
  E_PROGRESS.WAITING:
    _eres                   := Home(
                                    Execute   := TRUE,
                                    Position  := _HomeParameter^[_nAxisIndex].stHomingParam.Position,
                                    HomingMode:= _HomeParameter^[_nAxisIndex].stHomingParam.HomingMode,
                                    Options   := _HomeParameter^[_nAxisIndex].stHomingParam.Options);

    IF (_eres = E_PROGRESS.ERROR)
    THEN
      _eState               := E_PROGRESS.ERROR;
    ELSIF (_eres = E_PROGRESS.DONE)
    THEN
      _eState               := E_PROGRESS.WORKING;
    END_IF
END_CASE
CASE _eState
OF
  E_PROGRESS.WORKING:
    _eState                 := E_PROGRESS.DONE;

    _eres                   := Home(
                                    Execute   := FALSE,
                                    Position  := _HomeParameter^[_nAxisIndex].stHomingParam.Position,
                                    HomingMode:= _HomeParameter^[_nAxisIndex].stHomingParam.HomingMode,
                                    Options   := _HomeParameter^[_nAxisIndex].stHomingParam.Options);
END_CASE

AxisHome := _eState;
END_METHOD

METHOD AxisIdle : E_PROGRESS
VAR_INPUT
  Execute           : BOOL;
END_VAR
VAR_INST
  _eResult,
  _eState           : E_PROGRESS;
  _stMsg            : ST_Message;
  _nRetry           : UINT;
END_VAR
IF NOT Check() THEN AxisIdle := E_PROGRESS.ERROR; return; END_IF
IF NOT Execute THEN _eState := E_PROGRESS.INIT; END_IF

CASE _eState
OF
  E_PROGRESS.INIT:
    IF Execute 
    THEN
      memset(ADR(_stMsg),0,SIZEOF(_stMsg));
      _nRetry                       := 0;
      _eResult                      := Reset(FALSE);
      _eState                       := E_PROGRESS.BUSY;
    END_IF
END_CASE
CASE _eState
OF
  E_PROGRESS.BUSY:
    _eResult                        := Reset(TRUE);

    IF (_eResult = E_PROGRESS.DONE)
    THEN
      _nRetry                       := _nRetry + 1;
      _eState                       := E_PROGRESS.STARTUP;
    END_IF
END_CASE
CASE _eState
OF
  E_PROGRESS.STARTUP:
    _eResult                        := Reset(FALSE);
    _eResult                        := Enable(FALSE);
    _eState                         := E_PROGRESS.READY;
END_CASE
CASE _eState
OF
  E_PROGRESS.PREPARE:
    _eResult                        := Reset(FALSE);
    _eResult                        := Enable(FALSE);

    _eState                         := E_PROGRESS.BUSY;

    _stMsg.eType                    := E_MessageType.eMessageInfo;
    _stMsg.eDevice                  := e_Device.Axis + TO_DINT(_AxisRef.NcToPlc.AxisId);
    _stMsg.eSubdevice               :=  e_SubDevice.AxisControl_Enable;
    _stMsg.iErrorNumber             := _nErrorId;

    _stMsg.sText                    := concat(TO_STRING(_eCtrl), ' retry: ');
    _stMsg.sText                    := concat(_stMsg.sText, TO_STRING(_nRetry));

    f_MessageSet(_stMsg);
END_CASE
CASE _eState
OF
  E_PROGRESS.READY:
    _eResult                        := Enable(TRUE);

    IF (_nRetry > MAX_RETRY)
    THEN
      _eState                       := E_PROGRESS.ERROR;

    ELSIF (_eResult = E_PROGRESS.DONE)
    THEN
      Enable(FALSE);
      _eState                       := E_PROGRESS.DONE;

    ELSIF (_eResult = E_PROGRESS.ERROR)
    THEN
      _eState                       := E_PROGRESS.PREPARE;

      _nErrorId                     := _AxisRef.NcToPlc.ErrorCode;
    
      _stMsg.eType                  := E_MessageType.eMessageError;
      _stMsg.eDevice                := e_Device.Axis + TO_DINT(_AxisRef.NcToPlc.AxisId);
      _stMsg.eSubdevice             :=  e_SubDevice.AxisControl_Enable;
      _stMsg.iErrorNumber           := _nErrorId;

      _stMsg.sText                  := concat(TO_STRING(_eCtrl), ' error axis enable: ');
      _stMsg.sText                  := concat(_stMsg.sText, TO_STRING(_nAxisIndex));

      f_MessageSet(_stMsg);
    END_IF
END_CASE

AxisIdle                                := _eState;
END_METHOD

PROPERTY AxisIndex : uint
SET
END_SET
END_PROPERTY

PROPERTY AxisInfo : pointer to ARRAY[1..PLC_CONSTANT.MAX_AXIS] OF ST_AXIS_INFO
SET
_Info := AxisInfo;
END_SET
END_PROPERTY

METHOD PRIVATE AxisInit : E_PROGRESS
VAR_INPUT
  Execute           : BOOL;
END_VAR
VAR_INST
  _eResult,
  _eState           : E_PROGRESS;
  _rValue           : LREAL;
  _stMsg            : ST_Message;

  // access to CoE register
  _sDeviceName      : STRING(256) := 'NO NAME';
  _fbCoeRead				: Tc2_MC2_Drive.FB_CoERead;
END_VAR
IF NOT Check() THEN AxisInit := E_PROGRESS.ERROR; RETURN; END_IF
IF NOT Execute THEN _eState := E_PROGRESS.INIT; END_IF

CASE _eState
OF
  E_PROGRESS.INIT:
    IF Execute 
    THEN
      memset(ADR(_stMsg),0,SIZEOF(_stMsg));

      _nErrorId                     := 0;
      _rValue                       := 0;
      _eState                       := E_PROGRESS.BUSY;
      _eInit                        := _eState;
    END_IF
END_CASE
CASE _eState
OF
  E_PROGRESS.BUSY:
    _eState                         := E_PROGRESS.STARTUP;
    _eResult                        := StartUp(FALSE);
END_CASE
CASE _eState
OF
  E_PROGRESS.STARTUP:
    _eResult                        := StartUp(TRUE);
    IF (_eResult = E_PROGRESS.DONE)
    THEN
      _eState                       := E_PROGRESS.PREPARE;
      _eResult                      := AxisReset(FALSE);
    ELSIF (_eResult = E_PROGRESS.ERROR)
    THEN
      _eState                       := _eResult;

      _stMsg.eType                  := E_MessageType.eMessageError;
      _stMsg.eDevice                := e_Device.Axis + TO_DINT(_AxisRef.NcToPlc.AxisId);
      _stMsg.eSubdevice             := e_Subdevice.fbAxis_StartUp;
      _stMsg.iErrorNumber := _nErrorId  := 6666;

      _stMsg.sText                  := TO_STRING(_eState);
      f_MessageSet(_stMsg);

    END_IF
END_CASE
CASE _eState
OF
  E_PROGRESS.PREPARE:
    _eResult                        := AxisReset(TRUE);
    IF (_eResult = E_PROGRESS.DONE)
    THEN
      _fbCoeRead(
                Execute             := FALSE,
                NetId               := _AxisRef.ADS.NetId, 
                Axis                := _AxisRef);
  
      IF (EncoderType > 1)
      THEN
        memset(ADR(_sDeviceName),0,SIZEOF(_sDeviceName));
  
        _eState                     := E_PROGRESS.READY;
      ELSE
        _eState                     := E_PROGRESS.WORKING;
      END_IF
    ELSIF (_eResult = E_PROGRESS.ERROR)
    THEN
      _eState                       := _eResult;

      _stMsg.eType                  := E_MessageType.eMessageError;
      _stMsg.eDevice                := e_Device.Axis + TO_DINT(_AxisRef.NcToPlc.AxisId);
      _stMsg.eSubdevice             := e_Subdevice.fbAxis_StartupReset;
      _stMsg.iErrorNumber           := ErrorId;

      _stMsg.sText                  := TO_STRING(_eState);
      f_MessageSet(_stMsg);

    END_IF
END_CASE
CASE _eState
OF
  E_PROGRESS.READY:
    _eResult                        := AxisReset(FALSE);
    // get manufacturer device name in CoE
    _fbCoeRead.Index                := 16#1008;
    _fbCoeRead.SubIndex             := 0;
    _fbCoeRead.pDstBuf              := ADR(_sDeviceName);
    _fbCoeRead.BufLen               := SIZEOF(_sDeviceName);

    _fbCoeRead(
              Execute               := TRUE,
              NetId                 := _AxisRef.ADS.NetId, 
              Axis                  := _AxisRef);

    IF _fbCoeRead.Busy
    THEN
      _eState                       := E_PROGRESS.WAITING;
    END_IF
END_CASE
CASE _eState
OF
  E_PROGRESS.WAITING:
    _fbCoeRead(
              NetId                 := _AxisRef.ADS.NetId, 
              Axis                  := _AxisRef);

    IF NOT _fbCoeRead.Busy
    THEN
      _eState                       := E_PROGRESS.WORKING;
    END_IF

// in case encoder type is used without hardware, error must be ignored here
(*
    IF (_fbCoeRead.Error)
    THEN
      _eState                       := E_PROGRESS.ERROR;

      _Info^[_nAxisIndex].nErrorId  := SEL((_fbCoeRead.CANopenErrId > 0), _fbCoeRead.AdsErrId, _fbCoeRead.CANopenErrId);

      _stMsg.eType                  := E_MessageType.eMessageError;
      _stMsg.eDevice                := e_Device.Axis + TO_DINT(_AxisRef.NcToPlc.AxisId);
      _stMsg.eSubdevice             := e_Subdevice.fbCoeRead;

      _stMsg.iErrorNumber           := SEL((_fbCoeRead.CANopenErrId > 0), _fbCoeRead.AdsErrId, _fbCoeRead.CANopenErrId);

      _stMsg.sText                  := TO_STRING(_eState);
      f_MessageSet(_stMsg);

      _fbCoeRead(
                Execute             := FALSE,
                NetId               := _AxisRef.ADS.NetId, 
                Axis                := _AxisRef);

    ELSIF NOT _fbCoeRead.Busy
    THEN
      _eState                       := E_PROGRESS.WORKING;
    END_IF
*)
END_CASE
CASE _eState
OF
  E_PROGRESS.WORKING:
    _eState                         := E_PROGRESS.DONE;
    // set default for axis release
    AxisEnableNegative              := TRUE;
    AxisEnablePositive              := TRUE;

    // clear fb
    _fbCoeRead(
              Execute               := FALSE,
              NetId                 := _AxisRef.ADS.NetId, 
              Axis                  := _AxisRef);

    _stMsg.eType                    := E_MessageType.eMessageInfo;
    _stMsg.eDevice                  := e_Device.Axis + TO_DINT(_AxisRef.NcToPlc.AxisId);
    _stMsg.eSubdevice               := e_Subdevice.fbAxis_StartUp;
    _stMsg.iErrorNumber             := 0;
    _stMsg.sText                    := concat('Axis Init: ', TO_STRING(_eState));

    f_MessageSet(_stMsg);
END_CASE

AxisInit                            := _eState;
END_METHOD

METHOD AxisMoveToPosition : E_PROGRESS
VAR_INPUT
  Execute           : BOOL;
  Data              : ST_MOVE_DATA;
END_VAR
VAR_INST
  _eres,
  _eState           : E_PROGRESS;
END_VAR
IF NOT Check() THEN AxisMoveToPosition := E_PROGRESS.ERROR; RETURN; END_IF
IF NOT Execute THEN _eState := E_PROGRESS.INIT; END_IF

CASE _eState
OF
  E_PROGRESS.INIT:
    IF Execute 
    THEN
      _eState               := E_PROGRESS.BUSY;
    END_IF
END_CASE
CASE _eState
OF
  E_PROGRESS.BUSY:
    _eState                 := E_PROGRESS.WAITING;
    _eres                   := MoveToPos(
                                      Execute    := FALSE, 
                                      Position   := Data.rSetPos, 
                                      Vel        := Data.rSetVelo, 
                                      Acc        := Data.rAcc, 
                                      Dec        := Data.rDec, 
                                      Jerk       := Data.rJerk, 
                                      BufferMode := Tc2_MC2.MC_BufferMode.MC_Aborting);
END_CASE
CASE _eState
OF
  E_PROGRESS.WAITING:
    _eres                   := MoveToPos(
                                      Execute    := TRUE, 
                                      Position   := Data.rSetPos, 
                                      Vel        := Data.rSetVelo, 
                                      Acc        := Data.rAcc, 
                                      Dec        := Data.rDec, 
                                      Jerk       := Data.rJerk, 
                                      BufferMode := Tc2_MC2.MC_BufferMode.MC_Aborting);

    IF (_eres = E_PROGRESS.ERROR)
    THEN
        _eState             := E_PROGRESS.ERROR;
    ELSIF (_eres = E_PROGRESS.DONE)
    THEN 
      _eState               := E_PROGRESS.WORKING;
    END_IF
END_CASE
CASE _eState
OF
  E_PROGRESS.WORKING:
    _eState                 := E_PROGRESS.DONE;
    _eres                   := MoveToPos(
                                      Execute    := FALSE, 
                                      Position   := Data.rSetPos, 
                                      Vel        := Data.rSetVelo, 
                                      Acc        := Data.rAcc, 
                                      Dec        := Data.rDec, 
                                      Jerk       := Data.rJerk, 
                                      BufferMode := Tc2_MC2.MC_BufferMode.MC_Aborting);
END_CASE

AxisMoveToPosition := _eState;
END_METHOD

METHOD AxisMoveVelocity : E_PROGRESS
VAR_INPUT
  Execute           : BOOL;
  Data              : ST_MOVE_DATA;
END_VAR
VAR_INST
  _eres,
  _eState           : E_PROGRESS;
END_VAR
IF NOT Check() THEN AxisMoveVelocity := E_PROGRESS.ERROR; RETURN; END_IF
IF NOT Execute THEN _eState := E_PROGRESS.INIT; END_IF

CASE _eState
OF
  E_PROGRESS.INIT:
    IF Execute 
    THEN
      _eState               := E_PROGRESS.BUSY;
    END_IF
END_CASE
CASE _eState
OF
  E_PROGRESS.BUSY:
    _eState                 := E_PROGRESS.WAITING;
    _eres                   := MoveVelo(
                                    Execute     := FALSE, 
                                    Velocity    := Data.rSetVelo, 
                                    Acc         := Data.rAcc, 
                                    Dec         := Data.rDec, 
                                    Jerk        := Data.rJerk, 
                                    Direction   := Data.iDirection, 
                                    BufferMode  := Tc2_MC2.MC_BufferMode.MC_Aborting);
END_CASE
CASE _eState
OF
  E_PROGRESS.WAITING:
    _eres                   := MoveVelo(
                                    Execute     := TRUE, 
                                    Velocity    := Data.rSetVelo, 
                                    Acc         := Data.rAcc, 
                                    Dec         := Data.rDec, 
                                    Jerk        := Data.rJerk, 
                                    Direction   := Data.iDirection, 
                                    BufferMode  := Tc2_MC2.MC_BufferMode.MC_Aborting);
    IF (_eres = E_PROGRESS.ERROR)
    THEN
        _eState             := E_PROGRESS.ERROR;
    ELSIF (_eres = E_PROGRESS.DONE)
    THEN 
      _eState               := E_PROGRESS.WORKING;
    END_IF
END_CASE
CASE _eState
OF
  E_PROGRESS.WORKING:
    _eState                 := E_PROGRESS.DONE;
    _eres                   := MoveVelo(
                                    Execute     := FALSE, 
                                    Velocity    := Data.rSetVelo, 
                                    Acc         := Data.rAcc, 
                                    Dec         := Data.rDec, 
                                    Jerk        := Data.rJerk, 
                                    Direction   := Data.iDirection, 
                                    BufferMode  := Tc2_MC2.MC_BufferMode.MC_Aborting);
END_CASE

AxisMoveVelocity                := _eState;
END_METHOD

METHOD AxisParameterRead : E_PROGRESS
VAR_INPUT
  Execute           : BOOL;
  ParameterNr       : Tc2_MC2.MC_AxisParameter;
END_VAR
VAR_INST
  _eres,
  _eState           : E_PROGRESS;
  _rValue           : LREAL;
END_VAR
IF NOT Check() THEN AxisParameterRead := E_PROGRESS.ERROR; RETURN; END_IF
IF NOT Execute THEN _eState := E_PROGRESS.INIT; END_IF

CASE _eState
OF
  E_PROGRESS.INIT:
    IF Execute 
    THEN
      _rValue                                     := 0.0;
      _eState                                     := E_PROGRESS.BUSY;
    END_IF
END_CASE
CASE _eState
OF
  E_PROGRESS.BUSY:
    _eState                                       := E_PROGRESS.WAITING;
    _eres           := ReadParameter(
                                  Execute         := FALSE,
                                  ParameterNumber := ParameterNr);
END_CASE
CASE _eState
OF
  E_PROGRESS.WAITING:
    _eres           := ReadParameter(
                                  Execute         := TRUE,
                                  ParameterNumber := ParameterNr);

    IF (_eres = E_PROGRESS.ERROR)
    THEN
      _eState                                     := E_PROGRESS.ERROR;
    ELSIF (_eres = E_PROGRESS.DONE)
    THEN 
      _eState                                     := E_PROGRESS.WORKING;
    END_IF

  E_PROGRESS.WORKING:
    _eState                                       := E_PROGRESS.DONE;
    _eres           := ReadParameter(
                                  Execute         := FALSE,
                                  ParameterNumber := ParameterNr);

    _NcParameterWrt^[_nAxisIndex].rValue          :=
    _rParameterReadValue                          := 
    _rValue                                       :=ReadParameterValue;
END_CASE

AxisParameterRead := _eState;
END_METHOD

METHOD AxisParameterWrite : E_PROGRESS
VAR_INPUT
  Execute           : BOOL;
  ParameterNr       : Tc2_MC2.MC_AxisParameter;
END_VAR
VAR_INST
  _eres,
  _eState           : E_PROGRESS;
  _rValue           : LREAL;
END_VAR
IF NOT Check() THEN AxisParameterWrite := E_PROGRESS.ERROR; RETURN; END_IF
IF NOT Execute THEN _eState := E_PROGRESS.INIT; END_IF

CASE _eState
OF
  E_PROGRESS.INIT:
    IF Execute 
    THEN
      _rValue                                     := _NcParameterWrt^[_nAxisIndex].rValue;
      _eState                                     := E_PROGRESS.BUSY;
    END_IF
END_CASE
CASE _eState
OF
  E_PROGRESS.BUSY:
    _eState                                       := E_PROGRESS.WAITING;
    _eres           := WriteParameter(
                                  Execute         := FALSE,
                                  Value           := _rValue,
                                  ParameterNumber := ParameterNr);
END_CASE
CASE _eState
OF
  E_PROGRESS.WAITING:
    _eres           := WriteParameter(
                                  Execute         := TRUE,
                                  Value           := _rValue,
                                  ParameterNumber := ParameterNr);
    IF (_eres = E_PROGRESS.ERROR)
    THEN
      _eState                                     := E_PROGRESS.ERROR;
    ELSIF (_eres = E_PROGRESS.DONE)
    THEN 
      _eState                                     := E_PROGRESS.WORKING;
    END_IF

  E_PROGRESS.WORKING:
    _eState                                       := E_PROGRESS.DONE;
    _eres           := WriteParameter(
                                  Execute         := FALSE,
                                  Value           := _rValue,
                                  ParameterNumber := ParameterNr);
END_CASE

AxisParameterWrite                                    := _eState;
END_METHOD

METHOD AxisParameterWritePersistent : E_PROGRESS
VAR_INPUT
  Execute           : BOOL;
  ParameterNr       : Tc2_MC2.MC_AxisParameter;
END_VAR
VAR_INST
  _eres,
  _eState           : E_PROGRESS;
  _rValue           : LREAL;
END_VAR
IF NOT Check() THEN AxisParameterWritePersistent := E_PROGRESS.ERROR; RETURN; END_IF
IF NOT Execute THEN _eState := E_PROGRESS.INIT; END_IF

CASE _eState
OF
  E_PROGRESS.INIT:
    IF Execute 
    THEN
      _rValue                                     := _NcParameterWrt^[_nAxisIndex].rValue;
      _eState                                     := E_PROGRESS.BUSY;
    END_IF
END_CASE
CASE _eState
OF
  E_PROGRESS.BUSY:
    _eState                                       := E_PROGRESS.WAITING;
    _eres           := WriteParameterPersistent(
                                  Execute         := FALSE,
                                  Value           := _rValue,
                                  ParameterNumber := ParameterNr);
END_CASE
CASE _eState
OF
  E_PROGRESS.WAITING:
    _eres           := WriteParameterPersistent(
                                  Execute         := TRUE,
                                  Value           := _rValue,
                                  ParameterNumber := ParameterNr);
    IF (_eres = E_PROGRESS.ERROR)
    THEN
      _eState                                     := E_PROGRESS.ERROR;
    ELSIF (_eres = E_PROGRESS.DONE)
    THEN 
      _eState                                     := E_PROGRESS.WORKING;
    END_IF

  E_PROGRESS.WORKING:
    _eState                                       := E_PROGRESS.DONE;
    _eres           := WriteParameterPersistent(
                                  Execute         := FALSE,
                                  Value           := _rValue,
                                  ParameterNumber := ParameterNr);
END_CASE

AxisParameterWritePersistent                          := _eState;
END_METHOD

PROPERTY AxisRef : reference to Tc2_MC2.AXIS_REF
GET
AxisRef := _AxisRef;
END_GET
END_PROPERTY

METHOD AxisReset : E_PROGRESS
VAR_INPUT
  Execute           : BOOL;
END_VAR
VAR_INST
  _eres,
  _eState           : E_PROGRESS;
END_VAR
IF NOT Check() THEN AxisReset := E_PROGRESS.ERROR; RETURN; END_IF
IF NOT Execute THEN _eState := E_PROGRESS.INIT; END_IF

CASE _eState
OF
  E_PROGRESS.INIT:
    IF Execute 
    THEN
      _eState                       := E_PROGRESS.BUSY;
    END_IF
END_CASE
CASE _eState
OF
  E_PROGRESS.BUSY:
    _eres                           := Reset(FALSE);
    _eState                         := E_PROGRESS.WAITING;
END_CASE
CASE _eState
OF
  E_PROGRESS.WAITING:
    _eres                           := Reset(TRUE);
    IF (_eres = E_PROGRESS.DONE)
    THEN
      _eState                       := E_PROGRESS.WORKING;
    ELSIF (_eres = E_PROGRESS.ERROR)
    THEN
      _eState                       := E_PROGRESS.ERROR;
    END_IF
END_CASE
CASE _eState
OF
  E_PROGRESS.WORKING:
    _eres                           := Reset(FALSE);
    _eState                         := E_PROGRESS.DONE;
END_CASE

AxisReset                           := _eState;
END_METHOD

PROPERTY AxisState : pointer to ARRAY[1..PLC_CONSTANT.MAX_AXIS] OF ST_AXIS_STATE
SET
_State := AxisState;
END_SET
END_PROPERTY

METHOD AxisStop : E_PROGRESS
VAR_INPUT
  Execute           : BOOL;
  Data              : ST_MOVE_DATA;
END_VAR
VAR_INST
  _eres,
  _eState           : E_PROGRESS;
END_VAR
IF NOT Check() THEN AxisStop := E_PROGRESS.ERROR; RETURN; END_IF
IF NOT Execute THEN _eState := E_PROGRESS.INIT; END_IF

CASE _eState
OF
  E_PROGRESS.INIT:
    IF Execute 
    THEN
      _eState       := E_PROGRESS.BUSY;
    END_IF
END_CASE
CASE _eState
OF
  E_PROGRESS.BUSY:
    _eState         := E_PROGRESS.WAITING;
    _eres           := Stop(
                            Execute := FALSE, 
                            Dec     := Data.rDec, 
                            Jerk    := Data.rJerk);
END_CASE
CASE _eState
OF
  E_PROGRESS.WAITING:
    _eres           := Stop(
                            Execute := TRUE, 
                            Dec     := Data.rDec, 
                            Jerk    := Data.rJerk);

    IF (_eres = E_PROGRESS.ERROR)
    THEN
        _eState     := E_PROGRESS.ERROR;
    ELSIF (_eres = E_PROGRESS.DONE)
    THEN 
      _eState       := E_PROGRESS.WORKING;
    END_IF
END_CASE
CASE _eState
OF
  E_PROGRESS.WORKING:
    _eState         := E_PROGRESS.DONE;
    _eres           := Stop(
                            Execute := FALSE, 
                            Dec     := Data.rDec, 
                            Jerk    := Data.rJerk);
END_CASE

AxisStop := _eState;
END_METHOD

METHOD PRIVATE Check : BOOL
//-----------------------------------------------------------------------------
IF (_nAxisIndex < 1) OR
   (_nAxisIndex > PLC_CONSTANT.MAX_AXIS)
THEN
  _eCheck                 := E_CHECK_STATE.AXIS_INDEX_OUT_OF_RANGE;
  RETURN;
END_IF

IF NOT __ISVALIDREF(_Axes)
THEN
  _eCheck                 := E_CHECK_STATE.AXIS_REF_POINTER_INVALID;
  RETURN;
END_IF
//-----------------------------------------------------------------------------
// get my AXIS_REF pointer for use in base class
//-----------------------------------------------------------------------------
_AxisRef                  := _Axes[_nAxisIndex];
//-----------------------------------------------------------------------------

IF NOT (_Ctrl <> 0)
THEN
  _eCheck                 := E_CHECK_STATE.AXIS_CTRL_POINTER_INVALID;
  RETURN;
END_IF

IF NOT (_State <> 0)
THEN
  _eCheck                 := E_CHECK_STATE.AXIS_STATE_POINTER_INVALID;
  RETURN;
END_IF

IF NOT (_Info <> 0)
THEN
  _eCheck                 := E_CHECK_STATE.AXIS_INFO_POINTER_INVALID;
  RETURN;
END_IF

IF NOT (_Data <> 0)
THEN
  _eCheck                 := E_CHECK_STATE.AXIS_DATA_POINTER_INVALID;
  RETURN;
END_IF

IF NOT (_NcParameterWrt <> 0)
THEN
  _eCheck                 := E_CHECK_STATE.AXIS_NC_PARAMETER_POINTER_INVALID;
  RETURN;
END_IF

IF NOT (_NcParameterRd <> 0)
THEN
  _eCheck                 := E_CHECK_STATE.AXIS_NC_PARAMETER_POINTER_INVALID;
  RETURN;
END_IF

IF NOT (_HomeParameter <> 0)
THEN
  _eCheck                 := E_CHECK_STATE.AXIS_HOME_PARAMETER_POINTER_INVALID;
  RETURN;
END_IF

IF NOT (_GearInParameter <> 0)
THEN
  _eCheck                 := E_CHECK_STATE.AXIS_GEAR_IN_PARAMETER_POINTER_INVALID;
  RETURN;
END_IF
  
IF NOT (_MotionOptions <> 0)
THEN
  _eCheck                 := E_CHECK_STATE.AXIS_MOTION_OPTIONS_POINTER_INVALID;
  RETURN;
END_IF

//-----------------------------------------------------------------------------
//  NaN INF check
//-----------------------------------------------------------------------------
IF NOT IsFinite(F_LReal(_Data^[_nAxisIndex].rSetPos))
THEN
	_Data^[_nAxisIndex].rSetPos     := 0.0;
END_IF

IF NOT IsFinite(F_LReal(_Data^[_nAxisIndex].rSetVelo))
THEN
	_Data^[_nAxisIndex].rSetVelo    := 0.0;
END_IF

IF NOT IsFinite(F_LReal(_Data^[_nAxisIndex].rAcc))
THEN
	_Data^[_nAxisIndex].rAcc        := 0.0;
END_IF

IF NOT IsFinite(F_LReal(_Data^[_nAxisIndex].rDec))
THEN
	_Data^[_nAxisIndex].rDec        := 0.0;
END_IF

IF NOT IsFinite(F_LReal(_Data^[_nAxisIndex].rOverride))
THEN
	_Data^[_nAxisIndex].rOverride   := 0.0;
END_IF
//-----------------------------------------------------------------------------
//-----------------------------------------------------------------------------
_eCheck                   := E_CHECK_STATE.CHECK_DONE;
Check                     := TRUE;
//-----------------------------------------------------------------------------
//-----------------------------------------------------------------------------
END_METHOD

//-------------------------------------------------------------------------------------
//
//  HAUD 2024 01 20
//
//  Cmd
//    - gets state for ctrl
//    - checks for eInit to be done, before any other commands are accepted
//    - prepare your commands here
//    - init what you have to here
//
//-------------------------------------------------------------------------------------
METHOD PRIVATE Cmd  : E_AXIS_STATE
VAR_INPUT
  eCmd              : E_AXIS_CTRL;
END_VAR
VAR_INST
  _estate   : E_AXIS_STATE;
  _stMsg    : ST_Message;
END_VAR

CASE eCmd
OF
  //-------------------------------------------------------------------------------------
  E_AXIS_CTRL.AXIS_INIT:
    _eInit    := _eResult             := AxisInit(FALSE);
    _estate                           := E_AXIS_STATE.AXIS_INIT;
ELSE
  IF (_eInit <> E_PROGRESS.DONE)
  THEN
    _eResult                          := E_PROGRESS.INVALID;
    _estate                           := E_AXIS_STATE.AXIS_NO_INIT;
  ELSE
    CASE eCmd
    OF
      //---------------------------------------------------------------------------------
      E_AXIS_CTRL.AXIS_DISABLE:
        _eResult                      := AxisDisable(FALSE);
        _estate                       := E_AXIS_STATE.AXIS_DISABLE;

      //---------------------------------------------------------------------------------
      E_AXIS_CTRL.AXIS_ENABLE:
        _eResult                      := AxisEnable(FALSE);
        _estate                       := E_AXIS_STATE.AXIS_ENABLE;

      //---------------------------------------------------------------------------------
      E_AXIS_CTRL.AXIS_IDLE:
        _eResult                      := AxisIdle(FALSE);
        _estate                       := E_AXIS_STATE.AXIS_IDLE;

      //---------------------------------------------------------------------------------
      E_AXIS_CTRL.AXIS_HOME:
        _eResult                      := AxisHome(FALSE);
        _estate                       := E_AXIS_STATE.AXIS_HOME;

      //---------------------------------------------------------------------------------
      E_AXIS_CTRL.AXIS_MOVE_POS:
        _eResult                      := AxisMoveToPosition(FALSE, _Data^[_nAxisIndex]);
        _estate                       := E_AXIS_STATE.AXIS_MOVE_POS;

      //---------------------------------------------------------------------------------
      E_AXIS_CTRL.AXIS_MOVE_VELO:
        _eResult                      := AxisMoveVelocity(FALSE, _Data^[_nAxisIndex]);
        _estate                       := E_AXIS_STATE.AXIS_MOVE_VELO;

      //---------------------------------------------------------------------------------
      E_AXIS_CTRL.AXIS_RESET:
        // OnChange clear error bit
        _Info^[_nAxisIndex].bError    := FALSE;
        _eResult                      := AxisReset(FALSE);
        _estate                       := E_AXIS_STATE.AXIS_RESET;

      //---------------------------------------------------------------------------------
      E_AXIS_CTRL.AXIS_HALT:
        _eResult                      := AxisHalt(FALSE, _Data^[_nAxisIndex]);
        _estate                       := E_AXIS_STATE.AXIS_HALT;

      //---------------------------------------------------------------------------------
      E_AXIS_CTRL.AXIS_STOP:
        _eResult                      := AxisStop(FALSE, _Data^[_nAxisIndex]);
        _estate                       := E_AXIS_STATE.AXIS_STOP;


      //---------------------------------------------------------------------------------
      E_AXIS_CTRL.AXIS_MOVE_BUFFER:
        _eResult                      := AxisBufferPos(FALSE, _Data^[_nAxisIndex]);
        _estate                       := E_AXIS_STATE.AXIS_MOVE_BUFFER;


      //---------------------------------------------------------------------------------
      E_AXIS_CTRL.AXIS_MOVE_BUFFER_VELO:
        _eResult                      := AxisBufferVelo(FALSE, _Data^[_nAxisIndex]);
        _estate                       := E_AXIS_STATE.AXIS_MOVE_BUFFER_VELO;


      //---------------------------------------------------------------------------------
      E_AXIS_CTRL.AXIS_PARAMETER_READ:
        _eParameterNrRead             := _NcParameterRd^[_nAxisIndex].ParameterNumber;
        _eResult                      := AxisParameterRead(FALSE, _eParameterNrRead);
        _estate                       := E_AXIS_STATE.AXIS_PARAMETER_READ;


      //---------------------------------------------------------------------------------
      E_AXIS_CTRL.AXIS_PARAMETER_WRITE:
        _eParameterNrWrite            := _NcParameterWrt^[_nAxisIndex].ParameterNumber;
        _rParameterWrtValue           := _NcParameterWrt^[_nAxisIndex].rValue;
        _eResult                      := AxisParameterWrite(FALSE, _eParameterNrWrite);
        _estate                       := E_AXIS_STATE.AXIS_PARAMETER_WRITE;


      //---------------------------------------------------------------------------------
      E_AXIS_CTRL.AXIS_PARAMETER_WRITE_PERSISTENT:
        _eParameterNrWrite            := _NcParameterWrt^[_nAxisIndex].ParameterNumber;
        _rParameterWrtValue           := _NcParameterWrt^[_nAxisIndex].rValue;
        _eResult                      := AxisParameterWritePersistent(FALSE, _eParameterNrWrite);
        _estate                       := E_AXIS_STATE.AXIS_PARAMETER_WRITE_PERSISTENT;

      //---------------------------------------------------------------------------------
      E_AXIS_CTRL.AXIS_GEAR_IN:
        _eResult                      := AxisGearIn(FALSE);
        _estate                       := E_AXIS_STATE.AXIS_GEAR_IN;

      //---------------------------------------------------------------------------------    
      E_AXIS_CTRL.AXIS_GEAR_OUT:
        _eResult                      := AxisGearOut(FALSE);
        _estate                       := E_AXIS_STATE.AXIS_GEAR_OUT;

      //---------------------------------------------------------------------------------
      E_AXIS_CTRL.AXIS_GEAR_IN_MULTIMASTER:
        _fbGearInMultiMaster.Master1  := _MultiMasterDummyRef[1];
        _fbGearInMultiMaster.Master2  := _MultiMasterDummyRef[2];
        _fbGearInMultiMaster.Master3  := _MultiMasterDummyRef[3];
        _fbGearInMultiMaster.Master4  := _MultiMasterDummyRef[4];

        _eResult                      := AxisGearInMultiMaster(FALSE);
        _estate                       := E_AXIS_STATE.AXIS_GEAR_IN_MULTIMASTER;

    //-----------------------------------------------------------------------------------
    ELSE
      _estate                         := E_AXIS_STATE.AXIS_NULL;

      IF (eCmd = E_NCI_CTRL.NULL)
      THEN
        _eResult                      := E_PROGRESS.DONE;
      ELSE
        _eResult                      := E_PROGRESS.INVALID;
  
        _stMsg.eType                  := E_MessageType.eMessageError;
        _stMsg.eDevice                := E_Device.Axis + TO_DINT(_Axes[_nAxisIndex].NcToPlc.AxisId);
        _stMsg.eSubdevice             := e_Subdevice.AxisControl;
        _stMsg.iErrorNumber           := 0;
  
        _stMsg.sText                  := 'E_AXIS_CTRL.';
        _stMsg.sText                  := concat(_stMsg.sText, TO_STRING(eCmd));
        _stMsg.sText                  := concat(_stMsg.sText, ': ');
        _stMsg.sText                  := concat(_stMsg.sText, TO_STRING(_eResult));

        f_MessageSet(_stMsg);
      END_IF
    END_CASE
  END_IF // _eInit
END_CASE

Cmd                                   := _estate;
END_METHOD

METHOD PRIVATE GetCalibrationCam : BOOL
VAR_INST
  _bCal     : Bool;
END_VAR
IF NOT Check() THEN RETURN; END_IF

IF _HomeParameter^[_nAxisIndex].stHomingParam.SimulateHomeSensor
THEN
	IF (_AxisRef.NcToPlc.HomingState < 4)
  THEN
		_bCal := TRUE;
	ELSE
		_bCal := FALSE;
	END_IF
ELSIF _HomeParameter^[_nAxisIndex].stHomingParam.HomeOnLimitMin
THEN
	_bCal := _bLimitMin XOR _HomeParameter^[_nAxisIndex].stHomingParam.InvertHomeSensor;

ELSIF _HomeParameter^[_nAxisIndex].stHomingParam.HomeOnLimitMax
THEN
	_bCal := _bLimitMax XOR _HomeParameter^[_nAxisIndex].stHomingParam.InvertHomeSensor;
ELSE
	_bCal := _bCalibrationInput XOR _HomeParameter^[_nAxisIndex].stHomingParam.InvertHomeSensor;
END_IF

GetCalibrationCam := _bCal;
END_METHOD

PROPERTY HomingParameter : pointer to ARRAY[1..PLC_CONSTANT.MAX_AXIS] OF st_homing
SET
_HomeParameter := HomingParameter;
END_SET
END_PROPERTY

METHOD PRIVATE LogControl
VAR_INST
  _sResult,
  _sCtrl            : STRING(30);

  _stMsg            : ST_Message;
END_VAR
  _stMsg.eType               := E_MessageType.eMessageInfo;
  _stMsg.eDevice             := E_Device.Axis + TO_DINT(_AxisRef.NcToPlc.AxisId);
  _stMsg.eSubdevice          := e_Subdevice.AxisControl;
  _stMsg.iErrorNumber        := _nAxisIndex;

  _sCtrl                     := concat('E_AXIS_CTRL', '.');
  _sCtrl                     := concat(_sCtrl, TO_STRING(_eCtrl));

  _stMsg.sText               := concat('new command: ', _sCtrl);
  f_MessageSet(_stMsg);
END_METHOD

METHOD PRIVATE LogResult
VAR_INST
  _sResult,
  _sCtrl            : STRING(30);

  _stMsg            : ST_Message;
END_VAR

  _stMsg.eType               := E_MessageType.eMessageInfo;
  _stMsg.eDevice             := E_Device.Axis + TO_DINT(_AxisRef.NcToPlc.AxisId);
  _stMsg.eSubdevice          := e_Subdevice.AxisControl;
  _stMsg.iErrorNumber        := _nAxisIndex;

  _sCtrl                     := concat('E_AXIS_CTRL', '.');
  _sCtrl                     := concat(_sCtrl, TO_STRING(_eCtrl));

  _sResult                   := concat('E_PROGRESS', '.');
  _sResult                   := concat(_sResult, TO_STRING(_eResult));

  _stMsg.sText               := concat(_sCtrl, ' ');
  _stMsg.sText               := concat(_sCtrl, _sResult);
  f_MessageSet(_stMsg);
END_METHOD

PROPERTY MotionOptions : pointer to ARRAY[1..PLC_CONSTANT.MAX_AXIS] OF ST_MOTION_OPTIONS
SET
_MotionOptions := MotionOptions;
END_SET
END_PROPERTY

PROPERTY NcParameterValue : Lreal
GET
NcParameterValue := _rParameterReadValue;
END_GET
END_PROPERTY

PROPERTY ReadNcParameter : pointer to ARRAY[1..PLC_CONSTANT.MAX_AXIS] OF st_nc_parameter
SET
_NcParameterRd := ReadNcParameter;
END_SET
END_PROPERTY

METHOD PRIVATE ResetSoE : E_PROGRESS
VAR_INPUT
  Execute           : BOOL;
END_VAR
VAR_INST
  _eState           : E_PROGRESS;
  _rValue           : LREAL;
  _udiErrSer,
  _udiErrAds        : UDINT;
  _stMsg            : ST_Message;

	_fbReset		      : Tc2_MC2_Drive.FB_SoEReset;
  _tonDelay         : Tc2_Standard.TON;
	_nRepeat			    : UINT;

  _sErrorSercos     : Tc2_System.T_MaxString;

END_VAR
IF NOT Check() THEN ResetSoE := E_PROGRESS.ERROR; RETURN; END_IF
IF NOT Execute THEN _eState := E_PROGRESS.INIT; END_IF

CASE _eState
OF
  E_PROGRESS.INIT:
    IF Execute 
    THEN
      memset(ADR(_stMsg),0,SIZEOF(_stMsg));
      memset(ADR(_sErrorSercos),0,SIZEOF(_sErrorSercos));

		  _nRepeat                      := 1;
      _udiErrSer := _udiErrAds      := 0;
      _rValue                       := 0;
      _eState                       := E_PROGRESS.BUSY;
    END_IF
END_CASE
CASE _eState
OF
  E_PROGRESS.BUSY:
    _eState                         := E_PROGRESS.WAITING;
		_tonDelay(
            IN                      := FALSE);

		_fbReset(
            Execute                 := FALSE, 
            Timeout                 := T#2500MS, 
            Axis                    := _AxisRef);
END_CASE
CASE _eState
OF
  E_PROGRESS.WAITING:
		_tonDelay(
            PT                      := T#1500MS, 
            IN                      := TRUE);

		_fbReset(
            Execute                 := TRUE, 
            Axis                    := _AxisRef, 
            AdsErrId                => _udiErrAds, 
            SercosErrId             => _udiErrSer);

    IF _fbReset.Error
    THEN
      _stMsg.eType                  := E_MessageType.eMessageError;
      _stMsg.eDevice                := e_Device.Axis + TO_DINT(_AxisRef.NcToPlc.AxisId);
      _stMsg.eSubdevice             :=  e_SubDevice.fbResetSercos;
      _stMsg.iErrorNumber           := _udiErrAds;

      _sErrorSercos                 := Tc2_Utilities.DATA_TO_HEXSTR(ADR(_udiErrSer), SIZEOF(_udiErrSer), FALSE);

      _stMsg.sText                  := concat('Sercos Err Nr: ', _sErrorSercos);

      f_MessageSet(_stMsg);

      _Info^[_nAxisIndex].nErrorId := _udiErrSer;
      _eState                       := E_PROGRESS.ERROR;

		ELSIF NOT _fbReset.Busy
		THEN
      _eState                       := E_PROGRESS.WORKING;

    ELSE
      IF _tonDelay.Q AND
         _AxisRef.NcToPlc.StateDWord.28
      THEN
        _nRepeat                    := _nRepeat + 1;
        _eState                     := E_PROGRESS.BUSY;    
      END_IF

      IF (_nRepeat > 5)
      THEN
        _eState                     := E_PROGRESS.ERROR;
      END_IF
		END_IF
END_CASE
CASE _eState
OF
  E_PROGRESS.WORKING:
    _eState                         := E_PROGRESS.DONE;
END_CASE


ResetSoE := _eState;
END_METHOD

PROPERTY TargetWindow : lreal
GET
END_GET
SET
END_SET
END_PROPERTY

METHOD Template : E_PROGRESS
VAR_INPUT
  Execute           : BOOL;
END_VAR
VAR_INST
  _eState           : E_PROGRESS;
  _rValue           : LREAL;
  _udiErr           : UDINT;
  _stMsg            : ST_Message;


END_VAR
IF NOT Check() THEN _eState := E_PROGRESS.ERROR; END_IF
IF NOT Execute THEN _eState := E_PROGRESS.INIT; END_IF

CASE _eState
OF
  E_PROGRESS.INIT:
    IF Execute 
    THEN
      memset(ADR(_stMsg),0,SIZEOF(_stMsg));
      _udiErr                       := 0;
      _rValue                       := 0;
      _eState                       := E_PROGRESS.BUSY;
    END_IF
END_CASE
CASE _eState
OF
  E_PROGRESS.BUSY:
    _eState                         := E_PROGRESS.STARTUP;
END_CASE
CASE _eState
OF
  E_PROGRESS.STARTUP:
    _eState                         := E_PROGRESS.PREPARE;
END_CASE
CASE _eState
OF
  E_PROGRESS.PREPARE:
    _eState                         := E_PROGRESS.READY;
END_CASE
CASE _eState
OF
  E_PROGRESS.READY:
    _eState                         := E_PROGRESS.WAITING;
END_CASE
CASE _eState
OF
  E_PROGRESS.WAITING:
    _eState                         := E_PROGRESS.WORKING;
END_CASE
CASE _eState
OF
  E_PROGRESS.WORKING:
    _eState                         := E_PROGRESS.DONE;
END_CASE

Template_1 := _eState;
END_METHOD

PROPERTY WriteNcParameter : pointer to ARRAY[1..PLC_CONSTANT.MAX_AXIS] OF st_nc_parameter
SET
_NcParameterWrt := WriteNcParameter;
END_SET
END_PROPERTY

END_FUNCTION_BLOCK

(* stored: Version 1.1.0.1, ProductVersion 3.1.4024.12
   POU FB_McAxisCtrl: Id {999335a0-5af6-0c1d-15bd-a65b83fb504c}, SpecialFunc None
   Folder methods: Id {c0eb5de4-89eb-00eb-3204-efd0e884debd}
   Folder private: Id {72055c1e-ae08-0707-1b82-aa6a286c994c}
   Folder properties: Id {ec33a634-95a7-05e3-1cf2-1ebdb2bd51b4}
   Property Axes: Id {d1a038b3-28c4-0a30-3eec-6fb30703f53e}
   Set Set: Id {a34fa163-c682-0310-2adf-d8e91c170ae2}
   Method AxisBufferPos: Id {8bea1fe6-78db-0d06-2903-94e698371421}
   Method AxisBufferVelo: Id {374fe133-fb4a-0fd3-3a5b-fe68bfd11804}
   Property AxisCtrl: Id {6f4cd776-1490-073c-2411-2e9fa9e9a6b2}
   Set Set: Id {e630f942-2d4d-05b1-0f59-706c62e18b88}
   Property AxisData: Id {dd1871a7-f253-01d5-39fc-b8e8ee980c20}
   Set Set: Id {3a83fd26-6575-0237-0d2c-1c41a74f695f}
   Method AxisDisable: Id {5b07de5c-833d-0c24-00ad-ad559c3149a3}
   Method AxisEnable: Id {bdedff7a-4ac5-01d7-2a4e-56553b33f7f1}
   Method AxisGearIn: Id {93b372b7-90fa-0265-20ee-a1e0c6284158}
   Method AxisGearInMultiMaster: Id {2753b84c-8efc-02bd-1ed9-f32e456b6aa2}
   Property AxisGearInParameter: Id {b3665f5f-7d61-0534-18c3-fc4c139bfd64}
   Set Set: Id {c3054604-2569-09a1-2cae-8365cfdd1ede}
   Method AxisGearOut: Id {ecd7fdba-4017-0a44-19d0-26000bfe6621}
   Method AxisHalt: Id {9b3aecb2-f7be-0371-1558-f6e3e61aa21b}
   Method AxisHome: Id {4affed04-b463-0d9f-01c5-e55d9c21fdc1}
   Method AxisIdle: Id {91e094ba-3637-045f-257e-8b0236a82b6e}
   Property AxisIndex: Id {ec26ef16-42cd-03a5-0740-028e92c264af}
   Set Set: Id {72c20e5d-c07d-04e2-2e7f-3065a8d113f1}
   Property AxisInfo: Id {43262739-6eeb-0240-259b-c24a2b7c9b8b}
   Set Set: Id {9f325ee6-0044-0408-1b8f-3ba89b0236ae}
   Method AxisInit: Id {cfb847c0-d387-0e90-3f6c-326032cd73b0}
   Method AxisMoveToPosition: Id {27760da5-88ba-02a4-20e2-a43d8fea6b68}
   Method AxisMoveVelocity: Id {636baf69-d370-0962-3889-6678baa38f82}
   Method AxisParameterRead: Id {e888c5ae-12ad-0616-229c-9fc3342dcc87}
   Method AxisParameterWrite: Id {77ad02f2-e55b-0375-1054-18aeccc4f797}
   Method AxisParameterWritePersistent: Id {bfd2219d-61cd-01fc-2d61-aa05055375fb}
   Property AxisRef: Id {d622fbfb-1430-047a-062d-a4dac266c76c}
   Get Get: Id {47a12226-31e2-0390-1c5c-a7209008eb2f}
   Method AxisReset: Id {983134b4-72eb-0c42-3ead-aaa67397970d}
   Property AxisState: Id {3dca1f6c-4c2d-0a02-0ad3-e24fa848690b}
   Set Set: Id {03f024e1-d54b-0d56-094a-cef330b0eb6d}
   Method AxisStop: Id {4a327d1b-00a7-09b1-2b27-f1512672b30e}
   Method Check: Id {f8c19456-13e2-0915-179c-dd36c10cb739}
   Method Cmd: Id {1389b619-e85f-0feb-358b-830cf714b972}
   Method GetCalibrationCam: Id {cce8967b-3b33-0d3c-2e17-bfaefcd5c5f7}
   Property HomingParameter: Id {bbed7ae6-3372-0209-2101-be3ac0cae96a}
   Set Set: Id {2a0c1316-16a0-0fe7-392a-ae61fe490c44}
   Method LogControl: Id {d80366c5-11f3-0a8a-297c-4979ebf61c8a}
   Method LogResult: Id {6a095a86-ad22-09b9-1058-5124e0b4c567}
   Property MotionOptions: Id {923ce8f8-17ae-0577-329b-a9bd138026ab}
   Set Set: Id {3c68ebc7-a095-0efe-0dd0-71092a4ee16d}
   Property NcParameterValue: Id {4f83dc68-3391-08cc-2ba6-0dca5b6f9170}
   Get Get: Id {c17f1740-3dbe-0323-21bb-d695e230a5f7}
   Property ReadNcParameter: Id {73c29011-949c-0182-1bfa-4914a1c5e4f4}
   Set Set: Id {35143572-1cc0-0e7a-19af-74d16589d588}
   Method ResetSoE: Id {4d30f9e6-607e-0983-163c-f478b48c7089}
   Property TargetWindow: Id {11d68468-93e3-0097-23b1-e0b3bcb90db4}
   Get Get: Id {0f08b6bc-07d3-0b4c-37b4-d89d0cb7c963}
   Set Set: Id {57184c7f-cacd-0caa-26dc-e19203ff97eb}
   Method Template: Id {f7a6377b-3c3c-04fd-3517-7f39ac13b38f}
   Property WriteNcParameter: Id {a00e8910-77c8-0a98-3ecf-242a3b2549b9}
   Set Set: Id {15199a8a-b1d7-019e-133f-411483cbf6d2} *)
